# EPICS substitutions: EUROTHRM/EUROTHRM-IOC-01App/Db/devEurothrmA01.substitutions
# Note: this file is generated by generate_substitutions.py
file devEurothrm.template {
pattern { P, GAD, LAD, MODBUS_PV, MODBUS_SP, MODBUS_P, MODBUS_I, MODBUS_D, MODBUS_HS, MODBUS_LS, MODBUS_AT, MODBUS_HO, MODBUS_OP }
{ "\$(P)", "0", "1", "1", "2", "6", "8", "9", "111", "112", "270", "30", "3" }
}
